FUNCTION F_ITC_SendSDI : BOOL
(**************************************************************************************
 * 	Application		:	BoxControl Framework
 *	Revision		:	$Revision: 404529 $
 *	Revision date	:	$Date: 2018-04-23 08:21:38 +0200 (Mo., 23 Apr 2018) $
 *	Last changed by	:	$Author: b7bolm $
 *	URL				:	$URL: http://almscdc.swisslog.com/repo/SWPD/Development/BoxControlFramework/20_Release/trunk/01_Software/BCF/BCF/JumpStart/20_Product/10_App/11_Com/10_Lib/10_Conv/11_ITC/F_ITC_SendSDI.TcPOU $
 *
 *	Purpose			:	Wrap message - SIR
 *
 * ------------------------------------------------------------------------------------
 *	Copyright Swisslog [IP AG], Switzerland. All rights reserved.
 * 
 * ------------------------------------------------------------------------------------
 *	
 * 	Revision History: 
 *
 * 	VERSION			DATE			INITIALS			DESCRIPTION
 *	0.1				01.01.2001		swl					Example
 *
 **************************************************************************************)
VAR_INPUT
	eChannelSrc		: E_MFCS_Channel; // Source communicaton channel	
	SignalNumber	: INT; // Signal Number
	SignalState		: BOOL; // Signal Status
	eReturnCode		: E_ErrorConv; // Return code
END_VAR
VAR
	SDI				: ST_ITC_SDI; 
END_VAR

// Map values
SDI.SignalState := SignalState;
SDI.SignalNumber := SignalNumber;
SDI.ReturnCode := eReturnCode;

// Forward to ITC
F_ITC_SendSDI := fbITC_Manager.M_SendData(
					meChannel	:= eChannelSrc,
					mMsgType	:= E_ITC_MsgTypeConv.SEND_DIGITAL_INPUT,
					mpData		:= ADR(SDI),
					mLen		:= SIZEOF(SDI));

END_FUNCTION

(* stored: Version 1.1.0.1, ProductVersion 3.1.4022.12
   POU F_ITC_SendSDI: Id {9ad788ac-14f7-4bc6-a744-98123758e8fd}, SpecialFunc None *)
